// Implicitly generated code : DO NOT EDIT
FUNCTION CheckLRangeUnsigned : ULINT
VAR_INPUT
    value, lower, upper: ULINT;
END_VAR

// Implicitly generated code : Only an Implementation suggestion
{noflow}
IF (value < lower) THEN
    CheckLRangeUnsigned := lower;
ELSIF(value > upper) THEN
    CheckLRangeUnsigned := upper;
ELSE
    CheckLRangeUnsigned := value;
END_IF
{flow}

END_FUNCTION

(* stored: Version 1.1.0.1, ProductVersion 3.1.4022.18
   POU CheckLRangeUnsigned: Id {ae9aaa01-68d8-40a4-bee5-9d7e4bfe0b3a}, SpecialFunc CheckLRangeUnsigned *)
